
(* ===== HMI "HMI_RT_4" =====

HMI tags "EdgePowerLogicTags"
   "I1" : Real, internal
   "I2" : Real, internal
   "I3" : Real, internal
   "I_Avg" : Real, internal
   "L1_L2" : Real, internal
   "L2_L3" : Real, internal
   "L3_L1" : Real, internal
   "LL_Avg" : Real, internal
   "L1_N" : Real, internal
   "L2_N" : Real, internal
   "L3_N" : Real, internal
   "LN_Avg" : Real, internal
   "Ip_Address" : WString[254], internal
   "Port_Number" : WString[254], internal
   "Enable" : Bool, internal
   "Active_Power_Ph1" : Real, internal
   "Active_Power_Ph2" : Real, internal
   "Active_Power_Ph3" : Real, internal
   "Active_Power_Tot" : Real, internal
   "Power_Factor" : Real, internal
   "Frequency" : Real, internal
   "Total_Active_Energy_Imported" : LReal, internal
   "Connection_State" : Int, internal
*)